PROGRAM prgSimple
VAR
	_counter : ULINT;
	_counterActive : BOOL;
	_reset : BOOL;
END_VAR

IF(_counterActive) THEN _counter := _counter + 1; END_IF
IF(_reset) THEN _counter := 0; _reset := false; END_IF;

END_PROGRAM

(* stored: Version 1.1.0.1, ProductVersion 3.1.4024.2
   POU prgSimple: Id {5077cfbc-288b-4c64-97b4-c087f2bac30f}, SpecialFunc None *)
